FUNCTION_BLOCK ComposStartStop (* Composite Function Block Type *)
  (* Standard: 61499-2 *)
  (* Version 0.0, 18/05/2022, Admin, Schneider Electric, template *)
  PACKAGE Main;
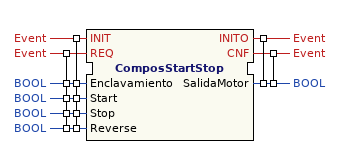
  EVENT_INPUT
    INIT WITH Enclavamiento, Start, Stop, Reverse; (* Initialization Request *)
    REQ WITH Enclavamiento, Start, Stop, Reverse; (* Normal Execution Request *)
  END_EVENT
  EVENT_OUTPUT
    INITO WITH SalidaMotor; (* Initialization Confirm *)
    CNF WITH SalidaMotor; (* Execution Confirmation *)
  END_EVENT
  VAR_INPUT
    Enclavamiento : BOOL; (* Input event qualifier *)
    Start : BOOL;
    Stop : BOOL;
    Reverse : BOOL;
  END_VAR
  VAR_OUTPUT
    SalidaMotor : BOOL; (* Output event qualifier *)
  END_VAR
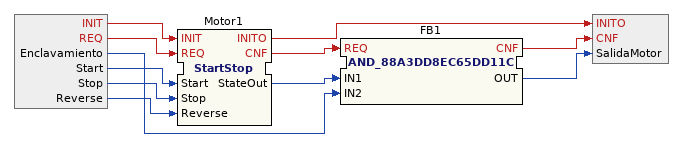
  FBS
    Motor1 : StartStop;
    FB1 : AND_88A3DD8EC65DD11C; {SET_ATTRIBUTE(Configuration.GenericFBType.InterfaceParams, Runtime.Standard#CNT:=2;OUT:BOOL)}
  END_FBS
  EVENT_CONNECTIONS
    INIT TO Motor1.INIT;
    REQ TO Motor1.REQ;
    Motor1.INITO TO INITO;
    FB1.CNF TO CNF;
    Motor1.CNF TO FB1.REQ;
  END_CONNECTIONS
  DATA_CONNECTIONS
    Motor1.StateOut TO FB1.IN1;
    Enclavamiento TO FB1.IN2;
    FB1.OUT TO SalidaMotor;
    Start TO Motor1.Start;
    Stop TO Motor1.Stop;
    Reverse TO Motor1.Reverse;
  END_CONNECTIONS
END_FUNCTION_BLOCK
